FUNCTION_BLOCK FB_RoofControl IMPLEMENTS I_Roof
VAR_INPUT
	min_speed				: UINT;			// minimum speed to drive
	max_speed				: UINT;			// maximum speed to drive
	acceleration			: UINT;			// acceleration [speed/call]
	max_position_diff		: INT;			// maximum allowed position difference between two drives of roof
	limit_slowdown			: REAL := 5;	// linear slowdown when moving towards limits starting at <x% and >(100-x)%
	min_position_1			: INT := 0;		// minimum position of roof
	max_position_1			: INT := 200;		// maximum position of roof
	min_position_2			: INT := 0;		// minimum position of roof
	max_position_2			: INT := 200;		// maximum position of roof

	// commands for automatic roof controls
	open_roofs				: BOOL;
	close_roofs				: BOOL;
	stop_roofs				: BOOL;
	reset_roofs				: BOOL;	
	open_roof				: ARRAY[1..2] OF BOOL;
	close_roof				: ARRAY[1..2] OF BOOL;
	stop_roof				: ARRAY[1..2] OF BOOL;
	reset_roof				: ARRAY[1..2] OF BOOL;
	
	// automatic mode
	automatic		AT%I*	: BOOL;
	
	// UPS failure
	ups_fail		AT%I*	: BOOL;
	
	// telemetry interval
	fTelemetryInterval		: TIME := T#5S;
END_VAR
VAR_OUTPUT
	// state
	roof_state				: E_RoofState;
	percent_open			: REAL;	
END_VAR
VAR
	// roofs
	roofs					: ARRAY[1..2] OF FB_Roof;
	
	// loop variable	
	i, j					: UINT;
	
	// open and close delays
	tonOpen2Delay			: TON;
	tonClose1Delay			: TON;
	
	// Comm
	fbComm					: I_Comm;	
	tonComm 				: TON;
	
	min_positions			: ARRAY[1..2] OF INT;		// minimum position of roof
	max_positions			: ARRAY[1..2] OF INT;		// maximum position of roof
END_VAR

// min_max
min_positions[1] := min_position_1;
max_positions[1] := max_position_1;
min_positions[2] := min_position_2;
max_positions[2] := max_position_2;

// call roofs
FOR i := 1 TO 2 DO
	// reset
	IF reset_roofs OR reset_roof[i] THEN
		roofs[i].Reset();
	END_IF	

	// automatic or manual mode
	IF automatic THEN
		roofs[i].Automatic(open_roof := open_roofs OR open_roof[i], close_roof := close_roofs OR close_roof[i], stop_roof := stop_roofs OR stop_roof[i]);
	ELSE
		roofs[i].Manual();
	END_IF

	// run 
	roofs[i](		
		roof_number			:= i,
		min_speed			:= min_speed,
		max_speed 			:= max_speed, 
		acceleration 		:= acceleration, 
		min_position 		:= min_positions[i], 
		max_position 		:= max_positions[i],
		max_position_diff 	:= max_position_diff,
		limit_slowdown		:= limit_slowdown,
		comm 				:= fbComm
	);
END_FOR

// set state
IF roofs[1].state = E_RoofState.error OR roofs[2].state = E_RoofState.error THEN
	roof_state := E_RoofState.error;
ELSIF roofs[1].state = E_RoofState.opened AND roofs[2].state = E_RoofState.opened THEN
	roof_state := E_RoofState.opened;
ELSIF roofs[1].state = E_RoofState.closed AND roofs[2].state = E_RoofState.closed THEN
	roof_state := E_RoofState.closed;
ELSIF roofs[1].state = E_RoofState.opening OR roofs[2].state = E_RoofState.opening THEN
	roof_state := E_RoofState.opening;	
ELSIF roofs[1].state = E_RoofState.closing OR roofs[2].state = E_RoofState.closing THEN
	roof_state := E_RoofState.closing;
ELSIF (roofs[1].state = E_RoofState.stopped OR roofs[1].state = E_RoofState.opened OR roofs[1].state = E_RoofState.closed) AND 
      (roofs[2].state = E_RoofState.stopped OR roofs[2].state = E_RoofState.opened OR roofs[2].state = E_RoofState.closed) THEN
	roof_state := E_RoofState.stopped;
ELSE
	roof_state := E_RoofState.error;	
END_IF

// percent open, clamped to 0..100: the over-travel margin and unsynced counters (after a restart with
// the roof halfway open) let the raw value leave that range, and telemetry uses -1.0 as the error marker.
// The per-roof values stay raw as a diagnostic of the counters.
percent_open := MAX(0.0, MIN(100.0, (roofs[1].percent_open + roofs[2].percent_open) / 2.0));

// send telemetry
tonComm(IN:=TRUE, PT:=fTelemetryInterval);
IF tonComm.Q THEN // publish new payload every fTelemetryInterval (default 5 seconds)
	tonComm(IN:=FALSE);
	THIS^._SendTelemetry();	
END_IF

METHOD _SendTelemetry : BOOL
VAR_INPUT
END_VAR
IF roof_state = E_RoofState.opened THEN
	fbComm.Publish('telescope', 'dome', 'AUXILIARY.DOME.REALPOS', '1.0');
ELSIF roof_state = E_RoofState.closed THEN
	fbComm.Publish('telescope', 'dome', 'AUXILIARY.DOME.REALPOS', '0.0');
ELSIF roof_state = E_RoofState.error THEN
	fbComm.Publish('telescope', 'dome', 'AUXILIARY.DOME.REALPOS', '-1.0');
ELSE
	fbComm.Publish('telescope', 'dome', 'AUXILIARY.DOME.REALPOS', LREAL_TO_STRING(percent_open / 100.0));
END_IF

IF roof_state = E_RoofState.opened OR roof_state = E_RoofState.opening THEN
	fbComm.Publish('telescope', 'dome', 'AUXILIARY.DOME.TARGETPOS', '1.0');
ELSIF roof_state = E_RoofState.closed OR roof_state = E_RoofState.closing THEN
	fbComm.Publish('telescope', 'dome', 'AUXILIARY.DOME.TARGETPOS', '0.0');
ELSIF roof_state = E_RoofState.stopped THEN
	fbComm.Publish('telescope', 'dome', 'AUXILIARY.DOME.TARGETPOS', LREAL_TO_STRING(percent_open / 100.0));
ELSE
	fbComm.Publish('telescope', 'dome', 'AUXILIARY.DOME.TARGETPOS', '-1.0');
END_IF

IF roof_state = E_RoofState.error THEN
	fbComm.Publish('telescope', 'dome', 'AUXILIARY.DOME.ERROR_STATE', '1');
	fbComm.Publish('telescope', 'dome', 'AUXILIARY.DOME.READY_STATE', '-1.0');
ELSE
	fbComm.Publish('telescope', 'dome', 'AUXILIARY.DOME.ERROR_STATE', '0');
	IF roof_state = E_RoofState.closed THEN
		fbComm.Publish('telescope', 'dome', 'AUXILIARY.DOME.READY_STATE', '0.0');
	ELSE
		fbComm.Publish('telescope', 'dome', 'AUXILIARY.DOME.READY_STATE', '1.0');
	END_IF
END_IF

IF state = E_RoofState.opening OR state = E_RoofState.closing THEN
	fbComm.Publish('telescope', 'dome', 'AUXILIARY.DOME.MOTION_STATE', '1.0');
ELSE
	fbComm.Publish('telescope', 'dome', 'AUXILIARY.DOME.MOTION_STATE', '0.0');
END_IF

// MONET specific
fbComm.Publish('telescope', 'dome', 'MONET.ROOF.STATE', Status);
fbComm.Publish('telescope', 'dome', 'MONET.ROOF.POS1', LREAL_TO_STRING(roofs[1].percent_open));
fbComm.Publish('telescope', 'dome', 'MONET.ROOF.STATE1', roofs[1].Status);
fbComm.Publish('telescope', 'dome', 'MONET.ROOF.ERROR1', roofs[1].Error);
fbComm.Publish('telescope', 'dome', 'MONET.ROOF.POS2', LREAL_TO_STRING(roofs[2].percent_open));
fbComm.Publish('telescope', 'dome', 'MONET.ROOF.STATE2', roofs[2].Status);
fbComm.Publish('telescope', 'dome', 'MONET.ROOF.ERROR2', roofs[2].Error);
END_METHOD

METHOD Close : BOOL
VAR_INPUT
END_VAR
FOR i := 1 TO 2 DO
	roofs[i].Close();
END_FOR;
END_METHOD

//FB_Init is always available implicitly and it is used primarily for initialization.
//The return value is not evaluated. For a specific influence, you can also declare the
//methods explicitly and provide additional code there with the standard initialization
//code. You can evaluate the return value.
METHOD FB_Init: BOOL
VAR_INPUT
    bInitRetains	: BOOL; // TRUE: the retain variables are initialized (reset warm / reset cold)
    bInCopyCode		: BOOL;  // TRUE: the instance will be copied to the copy code afterward (online change)
	comm			: I_Comm;   
END_VAR
THIS^.fbComm := comm;
END_METHOD

METHOD Open : BOOL
VAR_INPUT
END_VAR
FOR i := 1 TO 2 DO
	roofs[i].Open();
END_FOR;
END_METHOD

METHOD Reset : BOOL
VAR_INPUT
END_VAR
FOR i := 1 TO 2 DO
	roofs[i].Reset();
END_FOR;
END_METHOD

PROPERTY State : E_RoofState
GET
State := roof_state;
END_GET
END_PROPERTY

PROPERTY Status : STRING
GET
IF state = E_RoofState.closed THEN
	Status := 'CLOSED';
ELSIF state = E_RoofState.opened THEN
	Status := 'OPENED';
ELSIF state = E_RoofState.opening THEN
	Status := 'OPENING';
ELSIF state = E_RoofState.closing THEN
	Status := 'CLOSING';
ELSIF state = E_RoofState.stopped THEN
	Status := 'STOPPED';
ELSIF state = E_RoofState.error THEN
	Status := 'ERROR';
ELSIF state = E_RoofState.unknown THEN
	Status := 'UNKNOWN';	
END_IF
END_GET
END_PROPERTY

METHOD Stop : BOOL
VAR_INPUT
END_VAR
FOR i := 1 TO 2 DO
	roofs[i].Stop();
END_FOR;
END_METHOD

END_FUNCTION_BLOCK

(* stored: Version 1.1.0.1, ProductVersion 3.1.4024.15
   POU FB_RoofControl: Id {d87693f7-b561-4571-8c76-2cffdf8ef5fe}, SpecialFunc None
   Method _SendTelemetry: Id {35843360-1e80-4635-b873-96034fb47b44}
   Method Close: Id {09e5ef83-053e-434a-9daf-0f46715c9ca8}
   Method FB_Init: Id {dd850902-58ca-498a-b6a3-06589bee5a0c}
   Method Open: Id {158f37cb-bd12-4fa4-ba18-0d91b517278d}
   Method Reset: Id {e643a7f5-953f-43e5-b293-e4f6fb37cbd6}
   Property State: Id {7611ff11-7d75-4e77-a763-7a45ea36a762}
   Get Get: Id {63bdd3e1-4e74-409f-b6c0-a0531e107c7a}
   Property Status: Id {24fa5504-7504-4f2c-a2dc-6d5a61db8e4f}
   Get Get: Id {36e05c01-1ffa-42f8-87b2-d50fcb2efd5a}
   Method Stop: Id {b18a1fc2-196a-46c9-9a0b-0d399c89b25a} *)
